// TIA Portal V21 export
TYPE "lubricationSystemSta"
   STRUCT
      status : Struct
         ready : Bool;
         operation : Bool;
         run : Bool;
         alm : Bool;
         unackAlm : Bool;
         localMode : Bool;
         oilPump1Selected : Bool;
         oilPump2Selected : Bool;
         oilPreparationEn : Bool;
         flowSwitch : Bool;
         oilLevelMax : Bool;
         oilLevelMid : Bool;
         oilLevelMin : Bool;
         oilTempSwHigh : Bool;
         oilTempSwLow : Bool;
         heaterOn : Bool;
         waterVlvOpen : Bool;
         oilToCoolerVlv : Bool;
      END_STRUCT;
      statusDWord : DWord;
      "step" : USInt;
      stepTime : LTime;
      oilTempTank : Real;
      oilTempReturn : Real;
      oilFlow : Real;
      alm : "lubricationSystemAlm";
      almDWord : DWord;
      stopCtx : "lubricationSystemStopCtx";
   END_STRUCT;
END_TYPE
